RoboDK station: SandBox_UR5.rdk

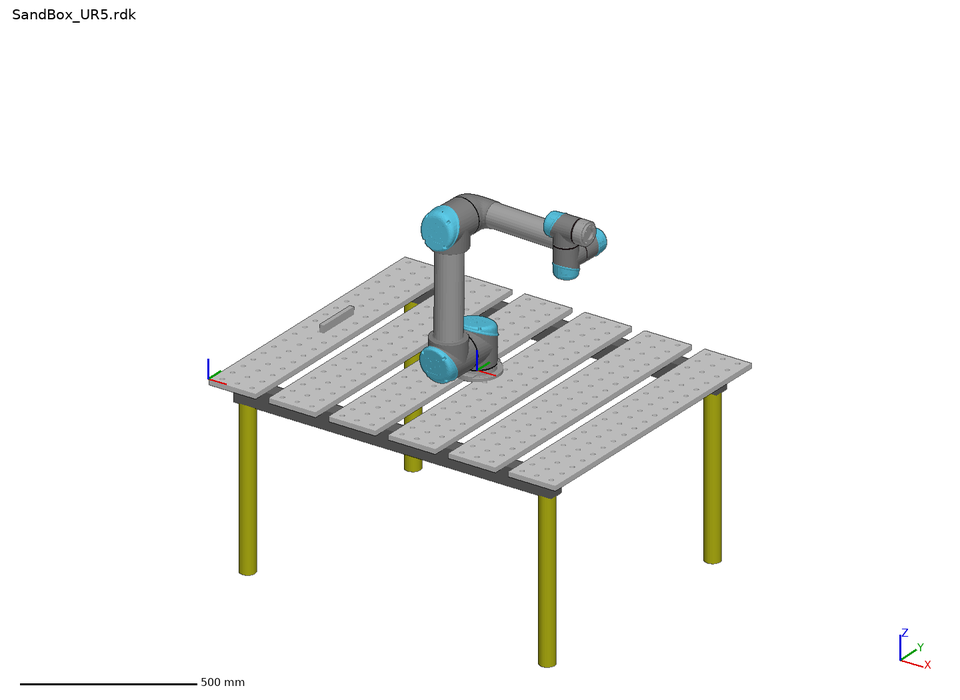
[picture v0: the station drawn from its stored meshes, robots at their saved joint values, targets as dots, program paths as lines]
Station SandBox_UR5 (saved by RoboDK 5.6.1). Poses are relative to the parent item; angles as X-Y-Z fixed-axis rotations.
  - frame UR5 Base at (0, 0, 0) mm
    - robot UR5: 6 axes
        modified DH rows (alpha deg, a mm, theta deg, d mm): 0, 0, 0, 89.2; 90, 0, 180, 0; 0, 425, 0, 0; 0, 392, 0, 109.3; -90, 0, 0, 94.75; 90, 0, 0, 82.5
        joint limits [-360, -360, -360, -360, -360, -360] to [360, 360, 360, 360, 360, 360]; home [0, -90, -90, 0, 90, 0]; saved at [-2.214, -90.7, -89.295, -0.005, 92.214, 0]
    - frame Table at (-590, -480, 0) mm
      - object part at (100, 500, 0) mm, rotated rx 0 ry 0 rz -90 deg, size 150 x 25 x 15 mm, geometry from part.stl
      - object table at (600, 480, 0) mm, size 1193.8 x 965.2 x 609.6 mm, geometry from welding_table.sld
